ABB RAPID module: Module1.mod

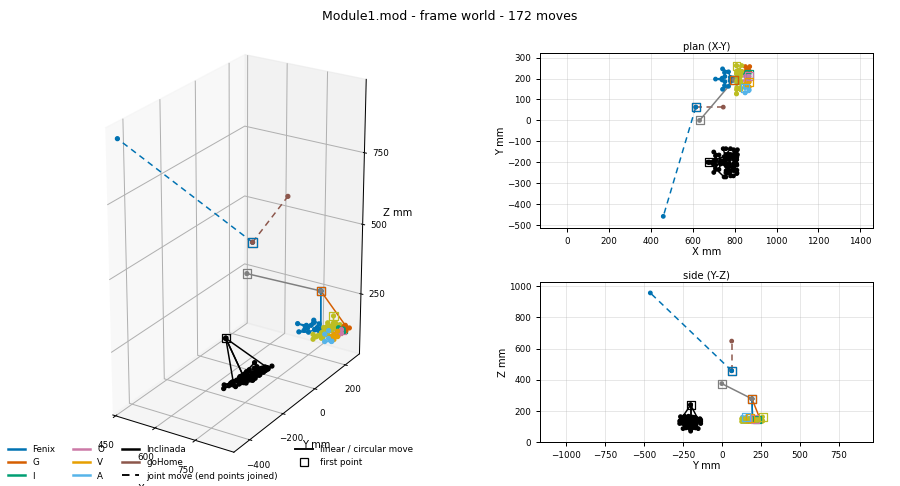
[picture p0: tool path of Module1.mod in frame world, 172 of 172 moves have a stored position in this frame; points joined in program order, loops and branches not executed]
MODULE Module1
    CONST robtarget Target_30:=[[-3.345189343,200,0],[0,0,1,0],[0,0,-1,1],[9E+09,9E+09,9E+09,9E+09,9E+09,9E+09]];
    CONST robtarget Target_20:=[[196.654810657,0,0],[0,0,1,0],[-1,-1,0,1],[9E+09,9E+09,9E+09,9E+09,9E+09,9E+09]];
    CONST robtarget Target_10:=[[811.652044776,0,588.439776326],[0.199367935,0,0.979924705,0],[0,0,0,0],[9E+09,9E+09,9E+09,9E+09,9E+09,9E+09]];
    CONST robtarget Target_40:=[[196.654810657,200,0],[0,0,1,0],[0,0,-1,1],[9E+09,9E+09,9E+09,9E+09,9E+09,9E+09]];
    CONST robtarget Target_50:=[[-3.345189343,0,0],[0,0,1,0],[-1,-1,0,1],[9E+09,9E+09,9E+09,9E+09,9E+09,9E+09]];
    CONST robtarget Home:=[[99.759101071,96.787006521,143.600305669],[0.000000093,0.707106794,-0.707106768,0.00000008],[0,-1,-1,0],[9E+09,9E+09,9E+09,9E+09,9E+09,9E+09]];
    CONST robtarget Target_110:=[[99.759,96.787,0],[0,-0.707106781,0.707106781,0],[0,-1,-1,0],[9E+09,9E+09,9E+09,9E+09,9E+09,9E+09]];
    CONST robtarget Target_140:=[[104.929185141,91.208348507,-1],[0,-0.707106781,0.707106781,0],[0,-1,-1,0],[9E+09,9E+09,9E+09,9E+09,9E+09,9E+09]];
    CONST robtarget Target_150:=[[107.828310564,78.545833086,-1],[0,-0.707106781,0.707106781,0],[0,-1,-1,0],[9E+09,9E+09,9E+09,9E+09,9E+09,9E+09]];
    CONST robtarget Target_160:=[[107.828310564,78.545833086,0],[0,-0.707106781,0.707106781,0],[0,-1,-1,0],[9E+09,9E+09,9E+09,9E+09,9E+09,9E+09]];
    CONST robtarget Target_170:=[[134.404345915,70.350066147,0],[0,-0.707106781,0.707106781,0],[0,-1,-1,0],[9E+09,9E+09,9E+09,9E+09,9E+09,9E+09]];
    CONST robtarget Target_180:=[[148.580115129,41.813525252,0],[0,-0.707106781,0.707106781,0],[0,-1,-1,0],[9E+09,9E+09,9E+09,9E+09,9E+09,9E+09]];
    CONST robtarget Target_190:=[[130.91133859,51.285461834,0],[0,-0.707106781,0.707106781,0],[0,-1,-1,0],[9E+09,9E+09,9E+09,9E+09,9E+09,9E+09]];
    CONST robtarget Target_200:=[[111.937087331,53.067189269,0],[0,-0.707106781,0.707106781,0],[0,-1,-1,0],[9E+09,9E+09,9E+09,9E+09,9E+09,9E+09]];
    CONST robtarget Target_210:=[[103.845690477,39.688183175,0],[0,-0.707106781,0.707106781,0],[0,-1,0,0],[9E+09,9E+09,9E+09,9E+09,9E+09,9E+09]];
    CONST robtarget Target_220:=[[99.759,8.211459743,0],[0,-0.707106781,0.707106781,0],[0,-1,0,0],[9E+09,9E+09,9E+09,9E+09,9E+09,9E+09]];
    CONST robtarget Target_230:=[[95.672309523,39.688183175,0],[0,-0.707106781,0.707106781,0],[0,-1,0,0],[9E+09,9E+09,9E+09,9E+09,9E+09,9E+09]];
    CONST robtarget Target_240:=[[87.580912669,53.067189269,0],[0,-0.707106781,0.707106781,0],[0,-1,0,0],[9E+09,9E+09,9E+09,9E+09,9E+09,9E+09]];
    CONST robtarget Target_250:=[[68.60666141,51.285461834,0],[0,-0.707106781,0.707106781,0],[0,-1,0,0],[9E+09,9E+09,9E+09,9E+09,9E+09,9E+09]];
    CONST robtarget Target_260:=[[50.937884871,41.813525252,0],[0,-0.707106781,0.707106781,0],[0,-1,0,0],[9E+09,9E+09,9E+09,9E+09,9E+09,9E+09]];
    CONST robtarget Target_270:=[[65.113654085,70.350066147,0],[0,-0.707106781,0.707106781,0],[0,-1,0,0],[9E+09,9E+09,9E+09,9E+09,9E+09,9E+09]];
    CONST robtarget Target_280:=[[91.689689436,78.545833086,0],[0,-0.707106781,0.707106781,0],[0,-1,-1,0],[9E+09,9E+09,9E+09,9E+09,9E+09,9E+09]];
    CONST robtarget Target_290:=[[94.588814859,91.208348507,0],[0,-0.707106781,0.707106781,0],[0,-1,-1,0],[9E+09,9E+09,9E+09,9E+09,9E+09,9E+09]];
    CONST robtarget Target_300:=[[99.759,96.787186115,0],[0,-0.707106781,0.707106781,0],[0,-1,-1,0],[9E+09,9E+09,9E+09,9E+09,9E+09,9E+09]];
    CONST robtarget Target_310:=[[51.434050484,162.594498178,0],[0,-0.707106781,0.707106781,0],[0,-1,-1,0],[9E+09,9E+09,9E+09,9E+09,9E+09,9E+09]];
    CONST robtarget Target_320:=[[64.567186307,162.594498178,0],[0,-0.707106781,0.707106781,0],[0,-1,-1,0],[9E+09,9E+09,9E+09,9E+09,9E+09,9E+09]];
    CONST robtarget Target_330:=[[63.433064042,150.856332741,0],[0,-0.707106781,0.707106781,0],[0,-1,-1,0],[9E+09,9E+09,9E+09,9E+09,9E+09,9E+09]];
    CONST robtarget Target_340:=[[40.013439281,150.867673964,0],[0,-0.707106781,0.707106781,0],[0,-1,-1,0],[9E+09,9E+09,9E+09,9E+09,9E+09,9E+09]];
    CONST robtarget Target_350:=[[40.013439281,171.554064067,0],[0,-0.707106781,0.707106781,0],[0,-1,-1,0],[9E+09,9E+09,9E+09,9E+09,9E+09,9E+09]];
    CONST robtarget Target_360:=[[63.410381597,171.588087735,0],[0,-0.707106781,0.707106781,0],[0,-1,-1,0],[9E+09,9E+09,9E+09,9E+09,9E+09,9E+09]];
    CONST robtarget Target_370:=[[64.567186307,167.539271251,0],[0,-0.707106781,0.707106781,0],[0,-1,-1,0],[9E+09,9E+09,9E+09,9E+09,9E+09,9E+09]];
    CONST robtarget Target_380:=[[67.932991772,167.539512506,10.290593582],[0.000000041,-0.707106747,0.707106815,0.000000103],[0,-1,-1,0],[9E+09,9E+09,9E+09,9E+09,9E+09,9E+09]];
    CONST robtarget Target_390:=[[73.897948354,167.539514704,10.290568716],[0.000000024,0.70710679,-0.707106772,-0.000000187],[0,-1,-1,0],[9E+09,9E+09,9E+09,9E+09,9E+09,9E+09]];
    CONST robtarget Target_410:=[[73.912353766,168.537298844,0],[0,-0.707106781,0.707106781,0],[0,-1,-1,0],[9E+09,9E+09,9E+09,9E+09,9E+09,9E+09]];
    CONST robtarget Target_400:=[[73.912353766,149.710869254,0],[0,-0.707106781,0.707106781,0],[0,-1,-1,0],[9E+09,9E+09,9E+09,9E+09,9E+09,9E+09]];
    CONST robtarget Target_420:=[[73.912362356,149.710913626,10.190706901],[0.000000042,0.707106789,-0.707106773,-0.000000141],[0,-1,-1,0],[9E+09,9E+09,9E+09,9E+09,9E+09,9E+09]];
    CONST robtarget Target_480:=[[86.637199295,167.641310207,13.160930267],[0.000000042,0.707106788,-0.707106775,-0.000000007],[0,-1,-1,0],[9E+09,9E+09,9E+09,9E+09,9E+09,9E+09]];
    CONST robtarget Target_470:=[[86.637205573,167.641342255,0],[0,-0.707106781,0.707106781,0],[0,-1,-1,0],[9E+09,9E+09,9E+09,9E+09,9E+09,9E+09]];
    CONST robtarget Target_440:=[[107.59578502,167.641342255,0],[0,-0.707106781,0.707106781,0],[0,-1,-1,0],[9E+09,9E+09,9E+09,9E+09,9E+09,9E+09]];
    CONST robtarget Target_450:=[[107.607126243,150.652190733,0],[0,-0.707106781,0.707106781,0],[0,-1,-1,0],[9E+09,9E+09,9E+09,9E+09,9E+09,9E+09]];
    CONST robtarget Target_460:=[[86.614523128,150.640849511,0],[0,-0.707106781,0.707106781,0],[0,-1,-1,0],[9E+09,9E+09,9E+09,9E+09,9E+09,9E+09]];
    CONST robtarget Target_530:=[[113.447892452,168.582709847,19.902538584],[0.000000053,0.707106797,-0.707106766,-0.000000049],[0,-1,-1,0],[9E+09,9E+09,9E+09,9E+09,9E+09,9E+09]];
    CONST robtarget Target_490:=[[113.447855905,168.582663735,0],[0,-0.707106781,0.707106781,0],[0,-1,-1,0],[9E+09,9E+09,9E+09,9E+09,9E+09,9E+09]];
    CONST robtarget Target_500:=[[124.335429644,149.710869254,0],[0,-0.707106781,0.707106781,0],[0,-1,-1,0],[9E+09,9E+09,9E+09,9E+09,9E+09,9E+09]];
    CONST robtarget Target_520:=[[127.035,149.711,0],[0,-0.707106781,0.707106781,0],[0,-1,-1,0],[9E+09,9E+09,9E+09,9E+09,9E+09,9E+09]];
    CONST robtarget Target_510:=[[137.377835685,168.582663735,0],[0,-0.707106781,0.707106781,0],[0,-1,-1,0],[9E+09,9E+09,9E+09,9E+09,9E+09,9E+09]];
    CONST robtarget Target_540:=[[137.377791379,168.582717891,19.385142962],[0.000000048,0.707106782,-0.70710678,-0.00000004],[0,-1,-1,0],[9E+09,9E+09,9E+09,9E+09,9E+09,9E+09]];
    CONST robtarget Target_590:=[[139.645827027,149.710937127,28.980061356],[-0.000000039,0.707106799,-0.707106764,-0.00000025],[0,-1,-1,0],[9E+09,9E+09,9E+09,9E+09,9E+09,9E+09]];
    CONST robtarget Target_550:=[[139.646080214,149.710869254,0],[0,-0.707106781,0.707106781,0],[0,-1,-1,0],[9E+09,9E+09,9E+09,9E+09,9E+09,9E+09]];
    CONST robtarget Target_560:=[[150.556336398,168.582663735,0],[0,-0.707106781,0.707106781,0],[0,-1,-1,0],[9E+09,9E+09,9E+09,9E+09,9E+09,9E+09]];
    CONST robtarget Target_570:=[[153.822608519,168.582663735,0],[0,-0.707106781,0.707106781,0],[0,-1,-1,0],[9E+09,9E+09,9E+09,9E+09,9E+09,9E+09]];
    CONST robtarget Target_580:=[[165.005054047,149.710869254,0],[0,-0.707106781,0.707106781,0],[0,-1,-1,0],[9E+09,9E+09,9E+09,9E+09,9E+09,9E+09]];
    CONST robtarget Target_600:=[[165.005120388,149.710943698,27.340042804],[0.000000095,0.707106812,-0.707106751,0.000000059],[0,-1,-1,0],[9E+09,9E+09,9E+09,9E+09,9E+09,9E+09]];
    CONST robtarget Home_3:=[[99.759101071,96.787006521,143.600305669],[0.000000093,0.707106794,-0.707106768,0.00000008],[1,1,0,7],[9E+09,9E+09,9E+09,9E+09,9E+09,9E+09]];
    CONST robtarget Target_110_3:=[[99.759,96.787,0],[0,-0.707106781,0.707106781,0],[1,1,-1,7],[9E+09,9E+09,9E+09,9E+09,9E+09,9E+09]];
    CONST robtarget Target_140_3:=[[104.929185141,91.208348507,-1],[0,-0.707106781,0.707106781,0],[1,1,-1,7],[9E+09,9E+09,9E+09,9E+09,9E+09,9E+09]];
    CONST robtarget Target_150_3:=[[107.828310564,78.545833086,-1],[0,-0.707106781,0.707106781,0],[1,1,-1,7],[9E+09,9E+09,9E+09,9E+09,9E+09,9E+09]];
    CONST robtarget Target_160_3:=[[107.828310564,78.545833086,0],[0,-0.707106781,0.707106781,0],[1,1,-1,7],[9E+09,9E+09,9E+09,9E+09,9E+09,9E+09]];
    CONST robtarget Target_170_3:=[[134.404345915,70.350066147,0],[0,-0.707106781,0.707106781,0],[1,1,-1,7],[9E+09,9E+09,9E+09,9E+09,9E+09,9E+09]];
    CONST robtarget Target_180_3:=[[148.580115129,41.813525252,0],[0,-0.707106781,0.707106781,0],[1,1,-1,7],[9E+09,9E+09,9E+09,9E+09,9E+09,9E+09]];
    CONST robtarget Target_190_3:=[[130.91133859,51.285461834,0],[0,-0.707106781,0.707106781,0],[1,1,-1,7],[9E+09,9E+09,9E+09,9E+09,9E+09,9E+09]];
    CONST robtarget Target_200_3:=[[111.937087331,53.067189269,0],[0,-0.707106781,0.707106781,0],[1,1,-1,7],[9E+09,9E+09,9E+09,9E+09,9E+09,9E+09]];
    CONST robtarget Target_210_3:=[[103.845690477,39.688183175,0],[0,-0.707106781,0.707106781,0],[1,1,-1,7],[9E+09,9E+09,9E+09,9E+09,9E+09,9E+09]];
    CONST robtarget Target_220_3:=[[99.759,8.211459743,0],[0,-0.707106781,0.707106781,0],[0,0,-1,7],[9E+09,9E+09,9E+09,9E+09,9E+09,9E+09]];
    CONST robtarget Target_230_3:=[[95.672309523,39.688183175,0],[0,-0.707106781,0.707106781,0],[1,1,-1,7],[9E+09,9E+09,9E+09,9E+09,9E+09,9E+09]];
    CONST robtarget Target_240_3:=[[87.580912669,53.067189269,0],[0,-0.707106781,0.707106781,0],[1,1,-1,7],[9E+09,9E+09,9E+09,9E+09,9E+09,9E+09]];
    CONST robtarget Target_250_3:=[[68.60666141,51.285461834,0],[0,-0.707106781,0.707106781,0],[1,1,-1,7],[9E+09,9E+09,9E+09,9E+09,9E+09,9E+09]];
    CONST robtarget Target_260_3:=[[50.937884871,41.813525252,0],[0,-0.707106781,0.707106781,0],[1,1,-1,7],[9E+09,9E+09,9E+09,9E+09,9E+09,9E+09]];
    CONST robtarget Target_270_3:=[[65.113654085,70.350066147,0],[0,-0.707106781,0.707106781,0],[1,1,-1,7],[9E+09,9E+09,9E+09,9E+09,9E+09,9E+09]];
    CONST robtarget Target_280_3:=[[91.689689436,78.545833086,0],[0,-0.707106781,0.707106781,0],[1,1,-1,7],[9E+09,9E+09,9E+09,9E+09,9E+09,9E+09]];
    CONST robtarget Target_290_3:=[[94.588814859,91.208348507,0],[0,-0.707106781,0.707106781,0],[1,1,-1,7],[9E+09,9E+09,9E+09,9E+09,9E+09,9E+09]];
    CONST robtarget Target_300_3:=[[99.759,96.787186115,0],[0,-0.707106781,0.707106781,0],[1,1,-1,7],[9E+09,9E+09,9E+09,9E+09,9E+09,9E+09]];
    CONST robtarget Target_310_3:=[[51.434050484,162.594498178,0],[0,-0.707106781,0.707106781,0],[1,1,-1,7],[9E+09,9E+09,9E+09,9E+09,9E+09,9E+09]];
    CONST robtarget Target_320_3:=[[64.567186307,162.594498178,0],[0,-0.707106781,0.707106781,0],[1,1,-1,7],[9E+09,9E+09,9E+09,9E+09,9E+09,9E+09]];
    CONST robtarget Target_330_3:=[[63.433064042,150.856332741,0],[0,-0.707106781,0.707106781,0],[1,1,-1,7],[9E+09,9E+09,9E+09,9E+09,9E+09,9E+09]];
    CONST robtarget Target_340_3:=[[40.013439281,150.867673964,0],[0,-0.707106781,0.707106781,0],[1,1,-1,7],[9E+09,9E+09,9E+09,9E+09,9E+09,9E+09]];
    CONST robtarget Target_350_3:=[[40.013439281,171.554064067,0],[0,-0.707106781,0.707106781,0],[1,1,-1,7],[9E+09,9E+09,9E+09,9E+09,9E+09,9E+09]];
    CONST robtarget Target_360_3:=[[63.410381597,171.588087735,0],[0,-0.707106781,0.707106781,0],[1,1,-1,7],[9E+09,9E+09,9E+09,9E+09,9E+09,9E+09]];
    CONST robtarget Target_370_3:=[[64.567186307,167.539271251,0],[0,-0.707106781,0.707106781,0],[1,1,-1,7],[9E+09,9E+09,9E+09,9E+09,9E+09,9E+09]];
    CONST robtarget Target_380_3:=[[67.932991772,167.539512506,10.290593582],[0.000000041,-0.707106747,0.707106815,0.000000103],[1,1,-1,7],[9E+09,9E+09,9E+09,9E+09,9E+09,9E+09]];
    CONST robtarget Target_390_3:=[[73.897948354,167.539514704,10.290568716],[0.000000024,0.70710679,-0.707106772,-0.000000187],[1,1,-1,7],[9E+09,9E+09,9E+09,9E+09,9E+09,9E+09]];
    CONST robtarget Target_410_3:=[[73.912353766,168.537298844,0],[0,-0.707106781,0.707106781,0],[1,1,-1,7],[9E+09,9E+09,9E+09,9E+09,9E+09,9E+09]];
    CONST robtarget Target_400_3:=[[73.912353766,149.710869254,0],[0,-0.707106781,0.707106781,0],[1,1,-1,7],[9E+09,9E+09,9E+09,9E+09,9E+09,9E+09]];
    CONST robtarget Target_420_3:=[[73.912362356,149.710913626,10.190706901],[0.000000042,0.707106789,-0.707106773,-0.000000141],[1,1,-1,7],[9E+09,9E+09,9E+09,9E+09,9E+09,9E+09]];
    CONST robtarget Target_480_3:=[[86.637199295,167.641310207,13.160930267],[0.000000042,0.707106788,-0.707106775,-0.000000007],[1,1,-1,7],[9E+09,9E+09,9E+09,9E+09,9E+09,9E+09]];
    CONST robtarget Target_470_3:=[[86.637205573,167.641342255,0],[0,-0.707106781,0.707106781,0],[1,1,-1,7],[9E+09,9E+09,9E+09,9E+09,9E+09,9E+09]];
    CONST robtarget Target_440_3:=[[107.59578502,167.641342255,0],[0,-0.707106781,0.707106781,0],[1,1,0,7],[9E+09,9E+09,9E+09,9E+09,9E+09,9E+09]];
    CONST robtarget Target_450_3:=[[107.607126243,150.652190733,0],[0,-0.707106781,0.707106781,0],[1,1,-1,7],[9E+09,9E+09,9E+09,9E+09,9E+09,9E+09]];
    CONST robtarget Target_460_3:=[[86.614523128,150.640849511,0],[0,-0.707106781,0.707106781,0],[1,1,-1,7],[9E+09,9E+09,9E+09,9E+09,9E+09,9E+09]];
    CONST robtarget Target_530_3:=[[113.447892452,168.582709847,19.902538584],[0.000000053,0.707106797,-0.707106766,-0.000000049],[1,1,0,7],[9E+09,9E+09,9E+09,9E+09,9E+09,9E+09]];
    CONST robtarget Target_490_3:=[[113.447855905,168.582663735,0],[0,-0.707106781,0.707106781,0],[1,1,0,7],[9E+09,9E+09,9E+09,9E+09,9E+09,9E+09]];
    CONST robtarget Target_500_3:=[[124.335429644,149.710869254,0],[0,-0.707106781,0.707106781,0],[1,1,0,7],[9E+09,9E+09,9E+09,9E+09,9E+09,9E+09]];
    CONST robtarget Target_520_3:=[[127.035,149.711,0],[0,-0.707106781,0.707106781,0],[1,1,0,7],[9E+09,9E+09,9E+09,9E+09,9E+09,9E+09]];
    CONST robtarget Target_510_3:=[[137.377835685,168.582663735,0],[0,-0.707106781,0.707106781,0],[1,1,0,7],[9E+09,9E+09,9E+09,9E+09,9E+09,9E+09]];
    CONST robtarget Target_540_3:=[[137.377791379,168.582717891,19.385142962],[0.000000048,0.707106782,-0.70710678,-0.00000004],[1,1,0,7],[9E+09,9E+09,9E+09,9E+09,9E+09,9E+09]];
    CONST robtarget Target_590_3:=[[139.645827027,149.710937127,28.980061356],[-0.000000039,0.707106799,-0.707106764,-0.00000025],[1,1,0,7],[9E+09,9E+09,9E+09,9E+09,9E+09,9E+09]];
    CONST robtarget Target_550_3:=[[139.646080214,149.710869254,0],[0,-0.707106781,0.707106781,0],[1,1,0,7],[9E+09,9E+09,9E+09,9E+09,9E+09,9E+09]];
    CONST robtarget Target_560_3:=[[150.556336398,168.582663735,0],[0,-0.707106781,0.707106781,0],[1,1,0,7],[9E+09,9E+09,9E+09,9E+09,9E+09,9E+09]];
    CONST robtarget Target_570_3:=[[153.822608519,168.582663735,0],[0,-0.707106781,0.707106781,0],[1,1,0,7],[9E+09,9E+09,9E+09,9E+09,9E+09,9E+09]];
    CONST robtarget Target_580_3:=[[165.005054047,149.710869254,0],[0,-0.707106781,0.707106781,0],[1,1,0,7],[9E+09,9E+09,9E+09,9E+09,9E+09,9E+09]];
    CONST robtarget Target_600_3:=[[165.005120388,149.710943698,27.340042804],[0.000000095,0.707106812,-0.707106751,0.000000059],[1,1,0,7],[9E+09,9E+09,9E+09,9E+09,9E+09,9E+09]];
    CONST robtarget Target_650:=[[631.875981178,0,375.874287303],[0.171236408,0,-0.985229969,0],[0,0,0,0],[9E+09,9E+09,9E+09,9E+09,9E+09,9E+09]];
    CONST robtarget Target_660:=[[35.046842978,108.443166881,26.254106583],[0,-0.707106781,0.707106781,0],[0,-1,-1,0],[9E+09,9E+09,9E+09,9E+09,9E+09,9E+09]];
    CONST robtarget Target_720:=[[35.047,108.443,0],[0,-0.707106781,0.707106781,0],[0,-1,-1,0],[9E+09,9E+09,9E+09,9E+09,9E+09,9E+09]];
    CONST robtarget Target_670:=[[35.046842978,133.443166881,0],[0,-0.707106781,0.707106781,0],[0,-1,-1,0],[9E+09,9E+09,9E+09,9E+09,9E+09,9E+09]];
    CONST robtarget Target_680:=[[56.373272958,116.727190549,0],[0,-0.707106781,0.707106781,0],[0,-1,-1,0],[9E+09,9E+09,9E+09,9E+09,9E+09,9E+09]];
    CONST robtarget Target_700:=[[62.660255206,108.443166881,0],[0,-0.707106781,0.707106781,0],[0,-1,-1,0],[9E+09,9E+09,9E+09,9E+09,9E+09,9E+09]];
    CONST robtarget Target_690:=[[62.660255206,133.443166881,0],[0,-0.707106781,0.707106781,0],[0,-1,-1,0],[9E+09,9E+09,9E+09,9E+09,9E+09,9E+09]];
    CONST robtarget Target_710:=[[62.660295778,133.257702122,17.408483113],[0.000000021,-0.707106766,0.707106797,0.000000049],[0,-1,-1,0],[9E+09,9E+09,9E+09,9E+09,9E+09,9E+09]];
    CONST robtarget Target_750:=[[73.779599663,128.906804208,17.663729092],[0.000000032,-0.70710677,0.707106793,0.000000042],[0,-1,-1,0],[9E+09,9E+09,9E+09,9E+09,9E+09,9E+09]];
    CONST robtarget Target_740:=[[73.779584595,128.906677729,0],[0,-0.707106781,0.707106781,0],[0,-1,-1,0],[9E+09,9E+09,9E+09,9E+09,9E+09,9E+09]];
    CONST robtarget Target_730:=[[73.779584595,108.443166881,0],[0,-0.707106781,0.707106781,0],[0,-1,-1,0],[9E+09,9E+09,9E+09,9E+09,9E+09,9E+09]];
    CONST robtarget Target_760:=[[73.779598222,108.443224437,17.731547844],[0.000000044,0.707106796,-0.707106766,-0.000000021],[0,-1,-1,0],[9E+09,9E+09,9E+09,9E+09,9E+09,9E+09]];
    CONST robtarget Target_830:=[[108.64148442,113.300223581,16.844032683],[0.000000008,0.707106783,-0.707106779,-0.000000028],[0,-1,-1,0],[9E+09,9E+09,9E+09,9E+09,9E+09,9E+09]];
    CONST robtarget Target_770:=[[108.641517534,113.300168853,0],[0,-0.707106781,0.707106781,0],[0,-1,-1,0],[9E+09,9E+09,9E+09,9E+09,9E+09,9E+09]];
    CONST robtarget Target_780:=[[107.593687159,109.466342423,0],[0,-0.707106781,0.707106781,0],[0,-1,-1,0],[9E+09,9E+09,9E+09,9E+09,9E+09,9E+09]];
    CONST robtarget Target_790:=[[87.573963293,109.429360175,0],[0,-0.707106781,0.707106781,0],[0,-1,-1,0],[9E+09,9E+09,9E+09,9E+09,9E+09,9E+09]];
    CONST robtarget Target_800:=[[87.586290709,127.945139267,0],[0,-0.707106781,0.707106781,0],[0,-1,-1,0],[9E+09,9E+09,9E+09,9E+09,9E+09,9E+09]];
    CONST robtarget Target_810:=[[107.593687159,127.932811851,0],[0,-0.707106781,0.707106781,0],[0,-1,-1,0],[9E+09,9E+09,9E+09,9E+09,9E+09,9E+09]];
    CONST robtarget Target_820:=[[108.641517534,124.074330589,0],[0,-0.707106781,0.707106781,0],[0,-1,-1,0],[9E+09,9E+09,9E+09,9E+09,9E+09,9E+09]];
    CONST robtarget Target_840:=[[108.641489854,124.074419597,17.530850048],[0.000000038,0.707106785,-0.707106778,-0.000000018],[0,-1,-1,0],[9E+09,9E+09,9E+09,9E+09,9E+09,9E+09]];
    CONST robtarget Target_900:=[[117.443278694,127.932797325,17.936531586],[-0.000000069,-0.707106731,0.707106831,0.000000105],[0,-1,-1,0],[9E+09,9E+09,9E+09,9E+09,9E+09,9E+09]];
    CONST robtarget Target_860:=[[117.443292682,127.932811851,0],[0,-0.707106781,0.707106781,0],[0,-1,-1,0],[9E+09,9E+09,9E+09,9E+09,9E+09,9E+09]];
    CONST robtarget Target_870:=[[140.224357771,127.932811851,0],[0,-0.707106781,0.707106781,0],[0,-1,-1,0],[9E+09,9E+09,9E+09,9E+09,9E+09,9E+09]];
    CONST robtarget Target_880:=[[140.236685187,109.466342423,0],[0,-0.707106781,0.707106781,0],[0,-1,-1,0],[9E+09,9E+09,9E+09,9E+09,9E+09,9E+09]];
    CONST robtarget Target_890:=[[117.418637849,109.454015007,0],[0,-0.707106781,0.707106781,0],[0,-1,-1,0],[9E+09,9E+09,9E+09,9E+09,9E+09,9E+09]];
    CONST robtarget Target_940:=[[150.283504114,128.956035202,17.783725507],[0,-0.707106781,0.707106781,0],[0,-1,-1,0],[9E+09,9E+09,9E+09,9E+09,9E+09,9E+09]];
    CONST robtarget Target_910:=[[150.283529368,128.955987394,0],[0,-0.707106781,0.707106781,0],[0,-1,-1,0],[9E+09,9E+09,9E+09,9E+09,9E+09,9E+09]];
    CONST robtarget Target_920:=[[150.283529368,108.443166881,0],[0,-0.707106781,0.707106781,0],[0,-1,-1,0],[9E+09,9E+09,9E+09,9E+09,9E+09,9E+09]];
    CONST robtarget Target_930:=[[170.106014575,108.443166881,0],[0,-0.707106781,0.707106781,0],[0,-1,-1,0],[9E+09,9E+09,9E+09,9E+09,9E+09,9E+09]];
    CONST robtarget Target_950:=[[170.105997965,108.443230949,17.745858799],[0.000000043,-0.707106776,0.707106786,0.000000052],[0,-1,-1,0],[9E+09,9E+09,9E+09,9E+09,9E+09,9E+09]];
    CONST robtarget Target_960:=[[51.434000123,162.594505433,12.553324918],[0.000000004,-0.707106757,0.707106805,0.000000033],[0,-1,-1,0],[9E+09,9E+09,9E+09,9E+09,9E+09,9E+09]];
    CONST robtarget Home_2:=[[99.759101071,96.787006521,143.600305669],[0.000000093,0.707106794,-0.707106768,0.00000008],[-1,-1,0,1],[9E+09,9E+09,9E+09,9E+09,9E+09,9E+09]];
    CONST robtarget Target_110_2:=[[99.759,96.787,0],[0,-0.707106781,0.707106781,0],[-1,-1,0,1],[9E+09,9E+09,9E+09,9E+09,9E+09,9E+09]];
    CONST robtarget Target_140_2:=[[104.929185141,91.208348507,-1],[0,-0.707106781,0.707106781,0],[-1,-1,0,1],[9E+09,9E+09,9E+09,9E+09,9E+09,9E+09]];
    CONST robtarget Target_150_2:=[[107.828310564,78.545833086,-1],[0,-0.707106781,0.707106781,0],[-1,-1,0,1],[9E+09,9E+09,9E+09,9E+09,9E+09,9E+09]];
    CONST robtarget Target_160_2:=[[107.828310564,78.545833086,0],[0,-0.707106781,0.707106781,0],[-1,-1,0,1],[9E+09,9E+09,9E+09,9E+09,9E+09,9E+09]];
    CONST robtarget Target_170_2:=[[134.404345915,70.350066147,0],[0,-0.707106781,0.707106781,0],[-1,-1,0,1],[9E+09,9E+09,9E+09,9E+09,9E+09,9E+09]];
    CONST robtarget Target_180_2:=[[148.580115129,41.813525252,0],[0,-0.707106781,0.707106781,0],[-1,-1,0,1],[9E+09,9E+09,9E+09,9E+09,9E+09,9E+09]];
    CONST robtarget Target_190_2:=[[130.91133859,51.285461834,0],[0,-0.707106781,0.707106781,0],[-1,-1,0,1],[9E+09,9E+09,9E+09,9E+09,9E+09,9E+09]];
    CONST robtarget Target_200_2:=[[111.937087331,53.067189269,0],[0,-0.707106781,0.707106781,0],[-1,-1,-1,1],[9E+09,9E+09,9E+09,9E+09,9E+09,9E+09]];
    CONST robtarget Target_210_2:=[[103.845690477,39.688183175,0],[0,-0.707106781,0.707106781,0],[-1,-1,-1,1],[9E+09,9E+09,9E+09,9E+09,9E+09,9E+09]];
    CONST robtarget Target_220_2:=[[99.759,8.211459743,0],[0,-0.707106781,0.707106781,0],[-1,-1,-1,1],[9E+09,9E+09,9E+09,9E+09,9E+09,9E+09]];
    CONST robtarget Target_230_2:=[[95.672309523,39.688183175,0],[0,-0.707106781,0.707106781,0],[-1,-1,-1,1],[9E+09,9E+09,9E+09,9E+09,9E+09,9E+09]];
    CONST robtarget Target_240_2:=[[87.580912669,53.067189269,0],[0,-0.707106781,0.707106781,0],[-1,-1,-1,1],[9E+09,9E+09,9E+09,9E+09,9E+09,9E+09]];
    CONST robtarget Target_250_2:=[[68.60666141,51.285461834,0],[0,-0.707106781,0.707106781,0],[-1,-1,-1,1],[9E+09,9E+09,9E+09,9E+09,9E+09,9E+09]];
    CONST robtarget Target_260_2:=[[50.937884871,41.813525252,0],[0,-0.707106781,0.707106781,0],[-1,-1,-1,1],[9E+09,9E+09,9E+09,9E+09,9E+09,9E+09]];
    CONST robtarget Target_270_2:=[[65.113654085,70.350066147,0],[0,-0.707106781,0.707106781,0],[-1,-1,-1,1],[9E+09,9E+09,9E+09,9E+09,9E+09,9E+09]];
    CONST robtarget Target_280_2:=[[91.689689436,78.545833086,0],[0,-0.707106781,0.707106781,0],[-1,-1,0,1],[9E+09,9E+09,9E+09,9E+09,9E+09,9E+09]];
    CONST robtarget Target_290_2:=[[94.588814859,91.208348507,0],[0,-0.707106781,0.707106781,0],[-1,-1,0,1],[9E+09,9E+09,9E+09,9E+09,9E+09,9E+09]];
    CONST robtarget Target_300_2:=[[99.759,96.787186115,0],[0,-0.707106781,0.707106781,0],[-1,-1,0,1],[9E+09,9E+09,9E+09,9E+09,9E+09,9E+09]];
    CONST robtarget Target_310_2:=[[51.434050484,162.594498178,0],[0,-0.707106781,0.707106781,0],[-1,-1,0,1],[9E+09,9E+09,9E+09,9E+09,9E+09,9E+09]];
    CONST robtarget Target_320_2:=[[64.567186307,162.594498178,0],[0,-0.707106781,0.707106781,0],[-1,-1,0,1],[9E+09,9E+09,9E+09,9E+09,9E+09,9E+09]];
    CONST robtarget Target_330_2:=[[63.433064042,150.856332741,0],[0,-0.707106781,0.707106781,0],[-1,-1,0,1],[9E+09,9E+09,9E+09,9E+09,9E+09,9E+09]];
    CONST robtarget Target_340_2:=[[40.013439281,150.867673964,0],[0,-0.707106781,0.707106781,0],[-1,-1,0,1],[9E+09,9E+09,9E+09,9E+09,9E+09,9E+09]];
    CONST robtarget Target_350_2:=[[40.013439281,171.554064067,0],[0,-0.707106781,0.707106781,0],[-1,-1,0,1],[9E+09,9E+09,9E+09,9E+09,9E+09,9E+09]];
    CONST robtarget Target_360_2:=[[63.410381597,171.588087735,0],[0,-0.707106781,0.707106781,0],[-1,-1,0,1],[9E+09,9E+09,9E+09,9E+09,9E+09,9E+09]];
    CONST robtarget Target_370_2:=[[64.567186307,167.539271251,0],[0,-0.707106781,0.707106781,0],[-1,-1,0,1],[9E+09,9E+09,9E+09,9E+09,9E+09,9E+09]];
    CONST robtarget Target_380_2:=[[67.932991772,167.539512506,10.290593582],[0.000000041,-0.707106747,0.707106815,0.000000103],[-1,-1,0,1],[9E+09,9E+09,9E+09,9E+09,9E+09,9E+09]];
    CONST robtarget Target_390_2:=[[73.897948354,167.539514704,10.290568716],[0.000000024,0.70710679,-0.707106772,-0.000000187],[-1,-1,0,1],[9E+09,9E+09,9E+09,9E+09,9E+09,9E+09]];
    CONST robtarget Target_410_2:=[[73.912353766,168.537298844,0],[0,-0.707106781,0.707106781,0],[-1,-1,0,1],[9E+09,9E+09,9E+09,9E+09,9E+09,9E+09]];
    CONST robtarget Target_400_2:=[[73.912353766,149.710869254,0],[0,-0.707106781,0.707106781,0],[-1,-1,0,1],[9E+09,9E+09,9E+09,9E+09,9E+09,9E+09]];
    CONST robtarget Target_420_2:=[[73.912362356,149.710913626,10.190706901],[0.000000042,0.707106789,-0.707106773,-0.000000141],[-1,-1,0,1],[9E+09,9E+09,9E+09,9E+09,9E+09,9E+09]];
    CONST robtarget Target_480_2:=[[86.637199295,167.641310207,13.160930267],[0.000000042,0.707106788,-0.707106775,-0.000000007],[-1,-1,0,1],[9E+09,9E+09,9E+09,9E+09,9E+09,9E+09]];
    CONST robtarget Target_470_2:=[[86.637205573,167.641342255,0],[0,-0.707106781,0.707106781,0],[-1,-1,0,1],[9E+09,9E+09,9E+09,9E+09,9E+09,9E+09]];
    CONST robtarget Target_440_2:=[[107.59578502,167.641342255,0],[0,-0.707106781,0.707106781,0],[-1,-1,0,1],[9E+09,9E+09,9E+09,9E+09,9E+09,9E+09]];
    CONST robtarget Target_450_2:=[[107.607126243,150.652190733,0],[0,-0.707106781,0.707106781,0],[-1,-1,0,1],[9E+09,9E+09,9E+09,9E+09,9E+09,9E+09]];
    CONST robtarget Target_460_2:=[[86.614523128,150.640849511,0],[0,-0.707106781,0.707106781,0],[-1,-1,0,1],[9E+09,9E+09,9E+09,9E+09,9E+09,9E+09]];
    CONST robtarget Target_530_2:=[[113.447892452,168.582709847,19.902538584],[0.000000053,0.707106797,-0.707106766,-0.000000049],[-1,-1,0,1],[9E+09,9E+09,9E+09,9E+09,9E+09,9E+09]];
    CONST robtarget Target_490_2:=[[113.447855905,168.582663735,0],[0,-0.707106781,0.707106781,0],[-1,-1,0,1],[9E+09,9E+09,9E+09,9E+09,9E+09,9E+09]];
    CONST robtarget Target_500_2:=[[124.335429644,149.710869254,0],[0,-0.707106781,0.707106781,0],[-1,-1,0,1],[9E+09,9E+09,9E+09,9E+09,9E+09,9E+09]];
    CONST robtarget Target_520_2:=[[127.035,149.711,0],[0,-0.707106781,0.707106781,0],[-1,-1,0,1],[9E+09,9E+09,9E+09,9E+09,9E+09,9E+09]];
    CONST robtarget Target_510_2:=[[137.377835685,168.582663735,0],[0,-0.707106781,0.707106781,0],[-1,-1,0,1],[9E+09,9E+09,9E+09,9E+09,9E+09,9E+09]];
    CONST robtarget Target_540_2:=[[137.377791379,168.582717891,19.385142962],[0.000000048,0.707106782,-0.70710678,-0.00000004],[-1,-1,0,1],[9E+09,9E+09,9E+09,9E+09,9E+09,9E+09]];
    CONST robtarget Target_590_2:=[[139.645827027,149.710937127,28.980061356],[-0.000000039,0.707106799,-0.707106764,-0.00000025],[-1,-1,0,1],[9E+09,9E+09,9E+09,9E+09,9E+09,9E+09]];
    CONST robtarget Target_550_2:=[[139.646080214,149.710869254,0],[0,-0.707106781,0.707106781,0],[-1,-1,0,1],[9E+09,9E+09,9E+09,9E+09,9E+09,9E+09]];
    CONST robtarget Target_560_2:=[[150.556336398,168.582663735,0],[0,-0.707106781,0.707106781,0],[-1,-1,0,1],[9E+09,9E+09,9E+09,9E+09,9E+09,9E+09]];
    CONST robtarget Target_570_2:=[[153.822608519,168.582663735,0],[0,-0.707106781,0.707106781,0],[-1,-1,0,1],[9E+09,9E+09,9E+09,9E+09,9E+09,9E+09]];
    CONST robtarget Target_580_2:=[[165.005054047,149.710869254,0],[0,-0.707106781,0.707106781,0],[-1,-1,0,1],[9E+09,9E+09,9E+09,9E+09,9E+09,9E+09]];
    CONST robtarget Target_600_2:=[[165.005120388,149.710943698,27.340042804],[0.000000095,0.707106812,-0.707106751,0.000000059],[-1,-1,0,1],[9E+09,9E+09,9E+09,9E+09,9E+09,9E+09]];
    CONST robtarget Target_660_2:=[[35.046842978,108.443166881,26.254106583],[0,-0.707106781,0.707106781,0],[-1,-1,0,1],[9E+09,9E+09,9E+09,9E+09,9E+09,9E+09]];
    CONST robtarget Target_720_2:=[[35.047,108.443,0],[0,-0.707106781,0.707106781,0],[-1,-1,0,1],[9E+09,9E+09,9E+09,9E+09,9E+09,9E+09]];
    CONST robtarget Target_670_2:=[[35.046842978,133.443166881,0],[0,-0.707106781,0.707106781,0],[-1,-1,0,1],[9E+09,9E+09,9E+09,9E+09,9E+09,9E+09]];
    CONST robtarget Target_700_2:=[[62.660255206,108.443166881,0],[0,-0.707106781,0.707106781,0],[-1,-1,0,1],[9E+09,9E+09,9E+09,9E+09,9E+09,9E+09]];
    CONST robtarget Target_690_2:=[[62.660255206,133.443166881,0],[0,-0.707106781,0.707106781,0],[-1,-1,0,1],[9E+09,9E+09,9E+09,9E+09,9E+09,9E+09]];
    CONST robtarget Target_710_2:=[[62.660295778,133.257702122,17.408483113],[0.000000021,-0.707106766,0.707106797,0.000000049],[-1,-1,0,1],[9E+09,9E+09,9E+09,9E+09,9E+09,9E+09]];
    CONST robtarget Target_750_2:=[[73.779599663,128.906804208,17.663729092],[0.000000032,-0.70710677,0.707106793,0.000000042],[-1,-1,0,1],[9E+09,9E+09,9E+09,9E+09,9E+09,9E+09]];
    CONST robtarget Target_740_2:=[[73.779584595,128.906677729,0],[0,-0.707106781,0.707106781,0],[-1,-1,0,1],[9E+09,9E+09,9E+09,9E+09,9E+09,9E+09]];
    CONST robtarget Target_730_2:=[[73.779584595,108.443166881,0],[0,-0.707106781,0.707106781,0],[-1,-1,0,1],[9E+09,9E+09,9E+09,9E+09,9E+09,9E+09]];
    CONST robtarget Target_760_2:=[[73.779598222,108.443224437,17.731547844],[0.000000044,0.707106796,-0.707106766,-0.000000021],[-1,-1,0,1],[9E+09,9E+09,9E+09,9E+09,9E+09,9E+09]];
    CONST robtarget Target_830_2:=[[108.64148442,113.300223581,16.844032683],[0.000000008,0.707106783,-0.707106779,-0.000000028],[-1,-1,0,1],[9E+09,9E+09,9E+09,9E+09,9E+09,9E+09]];
    CONST robtarget Target_770_2:=[[108.641517534,113.300168853,0],[0,-0.707106781,0.707106781,0],[-1,-1,0,1],[9E+09,9E+09,9E+09,9E+09,9E+09,9E+09]];
    CONST robtarget Target_780_2:=[[107.593687159,109.466342423,0],[0,-0.707106781,0.707106781,0],[-1,-1,0,1],[9E+09,9E+09,9E+09,9E+09,9E+09,9E+09]];
    CONST robtarget Target_790_2:=[[87.573963293,109.429360175,0],[0,-0.707106781,0.707106781,0],[-1,-1,0,1],[9E+09,9E+09,9E+09,9E+09,9E+09,9E+09]];
    CONST robtarget Target_800_2:=[[87.586290709,127.945139267,0],[0,-0.707106781,0.707106781,0],[-1,-1,0,1],[9E+09,9E+09,9E+09,9E+09,9E+09,9E+09]];
    CONST robtarget Target_810_2:=[[107.593687159,127.932811851,0],[0,-0.707106781,0.707106781,0],[-1,-1,0,1],[9E+09,9E+09,9E+09,9E+09,9E+09,9E+09]];
    CONST robtarget Target_820_2:=[[108.641517534,124.074330589,0],[0,-0.707106781,0.707106781,0],[-1,-1,0,1],[9E+09,9E+09,9E+09,9E+09,9E+09,9E+09]];
    CONST robtarget Target_840_2:=[[108.641489854,124.074419597,17.530850048],[0.000000038,0.707106785,-0.707106778,-0.000000018],[-1,-1,0,1],[9E+09,9E+09,9E+09,9E+09,9E+09,9E+09]];
    CONST robtarget Target_900_2:=[[117.443278694,127.932797325,17.936531586],[-0.000000069,-0.707106731,0.707106831,0.000000105],[-1,-1,0,1],[9E+09,9E+09,9E+09,9E+09,9E+09,9E+09]];
    CONST robtarget Target_860_3:=[[117.443292682,127.932811851,0],[0,-0.707106781,0.707106781,0],[-1,-1,0,1],[9E+09,9E+09,9E+09,9E+09,9E+09,9E+09]];
    CONST robtarget Target_870_2:=[[140.224357771,127.932811851,0],[0,-0.707106781,0.707106781,0],[-1,-1,0,1],[9E+09,9E+09,9E+09,9E+09,9E+09,9E+09]];
    CONST robtarget Target_880_2:=[[140.236685187,109.466342423,0],[0,-0.707106781,0.707106781,0],[-1,-1,0,1],[9E+09,9E+09,9E+09,9E+09,9E+09,9E+09]];
    CONST robtarget Target_890_2:=[[117.418637849,109.454015007,0],[0,-0.707106781,0.707106781,0],[-1,-1,0,1],[9E+09,9E+09,9E+09,9E+09,9E+09,9E+09]];
    CONST robtarget Target_940_2:=[[150.283504114,128.956035202,17.783725507],[0,-0.707106781,0.707106781,0],[-1,-1,0,1],[9E+09,9E+09,9E+09,9E+09,9E+09,9E+09]];
    CONST robtarget Target_910_2:=[[150.283529368,128.955987394,0],[0,-0.707106781,0.707106781,0],[-1,-1,0,1],[9E+09,9E+09,9E+09,9E+09,9E+09,9E+09]];
    CONST robtarget Target_920_2:=[[150.283529368,108.443166881,0],[0,-0.707106781,0.707106781,0],[-1,-1,0,1],[9E+09,9E+09,9E+09,9E+09,9E+09,9E+09]];
    CONST robtarget Target_930_2:=[[170.106014575,108.443166881,0],[0,-0.707106781,0.707106781,0],[-1,-1,0,1],[9E+09,9E+09,9E+09,9E+09,9E+09,9E+09]];
    CONST robtarget Target_950_2:=[[170.105997965,108.443230949,17.745858799],[0.000000043,-0.707106776,0.707106786,0.000000052],[-1,-1,0,1],[9E+09,9E+09,9E+09,9E+09,9E+09,9E+09]];
    CONST robtarget Target_980:=[[745.19998539,63.555998518,648.614999447],[0.403058195,0.127083777,0.864361092,0.272532031],[-1,0,0,0],[9E+09,9E+09,9E+09,9E+09,9E+09,9E+09]];
    TASK PERS wobjdata WorkPastel:=[FALSE,TRUE,"",[[700,297.348037667,137.083427328],[0.707046202,0.009255742,0.009255742,-0.707046202]],[[0,0,0],[1,0,0,0]]];
    TASK PERS wobjdata WorkPastel_2:=[FALSE,TRUE,"",[[663.397,-100,66.603],[0.683919377,0.179594782,-0.179594782,-0.683919377]],[[0,0,0],[1,0,0,0]]];
    CONST robtarget HomeRobot:=[[745.19998539,63.555998518,648.614999447],[0.403058195,0.127083777,0.864361092,0.272532031],[-1,0,0,0],[9E+09,9E+09,9E+09,9E+09,9E+09,9E+09]];
    CONST robtarget mantHerr:=[[494.621080465,494.792087576,971.864826811],[0.624444846,-0.306019376,0.699247952,0.165750044],[0,0,-1,0],[9E+09,9E+09,9E+09,9E+09,9E+09,9E+09]];
    CONST robtarget Target_970:=[[613.91794523,63.555999404,458.442114072],[0.041600547,0.221703595,0.952809214,0.203153911],[-1,0,0,0],[9E+09,9E+09,9E+09,9E+09,9E+09,9E+09]];
    CONST robtarget posMant:=[[458.575882142,-458.404912524,957.488606652],[0.61756941,0.262550436,0.653702432,-0.349783394],[-1,-1,-1,1],[9E+09,9E+09,9E+09,9E+09,9E+09,9E+09]];


!***********************************************************
    !
    ! M?dulo:  Module1
    !
    ! Descripción:
    !   <Introduzca la descripción aquí>
    !
    ! Autor: LENOVO
    !
    ! Versión: 1.0
    !
    !***********************************************************


    !***********************************************************
    !
    ! Procedimiento Main
    !
    !   Este es el punto de entrada de su programa
    !
    !***********************************************************
    PROC main()
        Inicio:
        IF DI_01=1 THEN
           Escribir;

        ENDIF
        IF DI_02=1 THEN
            Mantenimiento;
        ENDIF
        GOTO Inicio;
    ENDPROC

    LOCAL PROC Mantenimiento()
        Set DO_02;
        gomantHerr;
        Reset DO_02;
    ENDPROC

    LOCAL PROC Escribir()
        Set DO_01;
        goHome;
        goinicio;
        Fenix;
        Gio;
        Nic;
        goHome;
        Reset DO_01;
    ENDPROC

    LOCAL PROC Fenix()
        MoveL Home,v1000,z5,HerrG\WObj:=WorkPastel;
        MoveL Target_110,v500,z5,HerrG\WObj:=WorkPastel;
        MoveL Target_140,v100,z5,HerrG\WObj:=WorkPastel;
        MoveL Target_150,v100,z5,HerrG\WObj:=WorkPastel;
        MoveL Target_160,v100,z5,HerrG\WObj:=WorkPastel;
        MoveL Target_170,v100,z5,HerrG\WObj:=WorkPastel;
        MoveL Target_180,v100,z5,HerrG\WObj:=WorkPastel;
        MoveL Target_190,v100,z5,HerrG\WObj:=WorkPastel;
        MoveL Target_200,v100,z5,HerrG\WObj:=WorkPastel;
        MoveL Target_210,v100,z5,HerrG\WObj:=WorkPastel;
        MoveL Target_220,v100,z5,HerrG\WObj:=WorkPastel;
        MoveL Target_230,v100,z5,HerrG\WObj:=WorkPastel;
        MoveL Target_240,v100,z5,HerrG\WObj:=WorkPastel;
        MoveL Target_250,v100,z5,HerrG\WObj:=WorkPastel;
        MoveL Target_260,v100,z5,HerrG\WObj:=WorkPastel;
        MoveL Target_270,v100,z5,HerrG\WObj:=WorkPastel;
        MoveL Target_280,v100,z5,HerrG\WObj:=WorkPastel;
        MoveL Target_290,v100,z5,HerrG\WObj:=WorkPastel;
        MoveL Target_300,v100,z5,HerrG\WObj:=WorkPastel;
        MoveL Home,v500,z5,HerrG\WObj:=WorkPastel;
    ENDPROC
    LOCAL PROC G()
        MoveL Home,v1000,z5,HerrG\WObj:=WorkPastel;
        MoveL Target_960,v1000,z5,HerrG\WObj:=WorkPastel;
        MoveL Target_310,v100,z5,HerrG\WObj:=WorkPastel;
        MoveL Target_320,v100,z5,HerrG\WObj:=WorkPastel;
        MoveL Target_330,v100,z5,HerrG\WObj:=WorkPastel;
        MoveL Target_340,v100,z5,HerrG\WObj:=WorkPastel;
        MoveL Target_350,v100,z5,HerrG\WObj:=WorkPastel;
        MoveL Target_360,v100,z5,HerrG\WObj:=WorkPastel;
        MoveL Target_370,v100,z5,HerrG\WObj:=WorkPastel;
        MoveL Target_380,v100,z5,HerrG\WObj:=WorkPastel;
    ENDPROC
    LOCAL PROC I()
        MoveL Target_390,v100,z5,HerrG\WObj:=WorkPastel;
        MoveL Target_410,v100,z5,HerrG\WObj:=WorkPastel;
        MoveL Target_400,v100,z5,HerrG\WObj:=WorkPastel;
        MoveL Target_420,v100,z5,HerrG\WObj:=WorkPastel;
    ENDPROC
    LOCAL PROC O()
        MoveL Target_480,v100,z5,HerrG\WObj:=WorkPastel;
        MoveL Target_470,v100,z5,HerrG\WObj:=WorkPastel;
        MoveL Target_440,v100,z5,HerrG\WObj:=WorkPastel;
        MoveL Target_450,v100,z5,HerrG\WObj:=WorkPastel;
        MoveL Target_460,v100,z5,HerrG\WObj:=WorkPastel;
        MoveL Target_470,v100,z5,HerrG\WObj:=WorkPastel;
        MoveL Target_480,v100,z5,HerrG\WObj:=WorkPastel;
    ENDPROC
    LOCAL PROC V()
        MoveL Target_530,v100,z5,HerrG\WObj:=WorkPastel;
        MoveL Target_490,v100,z5,HerrG\WObj:=WorkPastel;
        MoveL Target_500,v100,z5,HerrG\WObj:=WorkPastel;
        MoveL Target_520,v100,z5,HerrG\WObj:=WorkPastel;
        MoveL Target_510,v100,z5,HerrG\WObj:=WorkPastel;
        MoveL Target_540,v100,z5,HerrG\WObj:=WorkPastel;
    ENDPROC
    LOCAL PROC A()
        MoveL Target_590,v1000,z5,HerrG\WObj:=WorkPastel;
        MoveL Target_550,v500,z5,HerrG\WObj:=WorkPastel;
        MoveL Target_560,v100,z5,HerrG\WObj:=WorkPastel;
        MoveL Target_570,v100,z5,HerrG\WObj:=WorkPastel;
        MoveL Target_580,v100,z5,HerrG\WObj:=WorkPastel;
        MoveL Target_600,v500,z5,HerrG\WObj:=WorkPastel;
    ENDPROC
    PROC Gio()
        G;
        I;
        O;
        V;
        A;
    ENDPROC
    PROC Inclinada()
        MoveJ Home_2,v1000,z5,HerrG\WObj:=WorkPastel_2;
        MoveL Target_110_2,v100,z5,HerrG\WObj:=WorkPastel_2;
        MoveL Target_140_2,v100,z5,HerrG\WObj:=WorkPastel_2;
        MoveL Target_150_2,v100,z5,HerrG\WObj:=WorkPastel_2;
        MoveL Target_160_2,v100,z5,HerrG\WObj:=WorkPastel_2;
        MoveL Target_170_2,v100,z5,HerrG\WObj:=WorkPastel_2;
        MoveL Target_180_2,v100,z5,HerrG\WObj:=WorkPastel_2;
        MoveL Target_190_2,v100,z5,HerrG\WObj:=WorkPastel_2;
        MoveL Target_200_2,v100,z5,HerrG\WObj:=WorkPastel_2;
        MoveL Target_210_2,v100,z5,HerrG\WObj:=WorkPastel_2;
        MoveL Target_220_2,v100,z5,HerrG\WObj:=WorkPastel_2;
        MoveL Target_230_2,v100,z5,HerrG\WObj:=WorkPastel_2;
        MoveL Target_240_2,v100,z5,HerrG\WObj:=WorkPastel_2;
        MoveL Target_250_2,v100,z5,HerrG\WObj:=WorkPastel_2;
        MoveL Target_260_2,v100,z5,HerrG\WObj:=WorkPastel_2;
        MoveL Target_270_2,v100,z5,HerrG\WObj:=WorkPastel_2;
        MoveL Target_280_2,v100,z5,HerrG\WObj:=WorkPastel_2;
        MoveL Target_290_2,v100,z5,HerrG\WObj:=WorkPastel_2;
        MoveL Target_300_2,v100,z5,HerrG\WObj:=WorkPastel_2;
        MoveL Home_2,v1000,z5,HerrG\WObj:=WorkPastel_2;
        MoveL Target_310_2,v100,z1,HerrG\WObj:=WorkPastel_2;
        MoveL Target_320_2,v100,z5,HerrG\WObj:=WorkPastel_2;
        MoveL Target_330_2,v100,z5,HerrG\WObj:=WorkPastel_2;
        MoveL Target_340_2,v100,z5,HerrG\WObj:=WorkPastel_2;
        MoveL Target_350_2,v100,z5,HerrG\WObj:=WorkPastel_2;
        MoveL Target_360_2,v100,z5,HerrG\WObj:=WorkPastel_2;
        MoveL Target_370_2,v100,z5,HerrG\WObj:=WorkPastel_2;
        MoveL Target_380_2,v100,z5,HerrG\WObj:=WorkPastel_2;
        MoveL Target_390_2,v100,z5,HerrG\WObj:=WorkPastel_2;
        MoveL Target_410_2,v100,z5,HerrG\WObj:=WorkPastel_2;
        MoveL Target_400_2,v100,z5,HerrG\WObj:=WorkPastel_2;
        MoveL Target_420_2,v100,z5,HerrG\WObj:=WorkPastel_2;
        MoveL Target_480_2,v100,z5,HerrG\WObj:=WorkPastel_2;
        MoveL Target_470_2,v100,z5,HerrG\WObj:=WorkPastel_2;
        MoveL Target_440_2,v100,z5,HerrG\WObj:=WorkPastel_2;
        MoveL Target_450_2,v100,z5,HerrG\WObj:=WorkPastel_2;
        MoveL Target_460_2,v100,z5,HerrG\WObj:=WorkPastel_2;
        MoveL Target_470_2,v100,z5,HerrG\WObj:=WorkPastel_2;
        MoveL Target_480_2,v100,z5,HerrG\WObj:=WorkPastel_2;
        MoveL Target_530_2,v100,z5,HerrG\WObj:=WorkPastel_2;
        MoveL Target_490_2,v100,z5,HerrG\WObj:=WorkPastel_2;
        MoveL Target_500_2,v100,z5,HerrG\WObj:=WorkPastel_2;
        MoveL Target_520_2,v100,z5,HerrG\WObj:=WorkPastel_2;
        MoveL Target_510_2,v100,z5,HerrG\WObj:=WorkPastel_2;
        MoveL Target_540_2,v100,z5,HerrG\WObj:=WorkPastel_2;
        MoveL Target_590_2,v100,z5,HerrG\WObj:=WorkPastel_2;
        MoveL Target_550_2,v100,z5,HerrG\WObj:=WorkPastel_2;
        MoveL Target_560_2,v100,z5,HerrG\WObj:=WorkPastel_2;
        MoveL Target_570_2,v100,z5,HerrG\WObj:=WorkPastel_2;
        MoveL Target_580_2,v100,z5,HerrG\WObj:=WorkPastel_2;
        MoveL Target_600_2,v100,z5,HerrG\WObj:=WorkPastel_2;
        MoveL Target_660_2,v100,z5,HerrG\WObj:=WorkPastel_2;
        MoveL Target_720_2,v100,z5,HerrG\WObj:=WorkPastel_2;
        MoveL Target_670_2,v100,z5,HerrG\WObj:=WorkPastel_2;
        MoveL Target_700_2,v100,z5,HerrG\WObj:=WorkPastel_2;
        MoveL Target_690_2,v100,z5,HerrG\WObj:=WorkPastel_2;
        MoveL Target_710_2,v100,z5,HerrG\WObj:=WorkPastel_2;
        MoveL Target_750_2,v100,z5,HerrG\WObj:=WorkPastel_2;
        MoveL Target_740_2,v100,z5,HerrG\WObj:=WorkPastel_2;
        MoveL Target_730_2,v100,z5,HerrG\WObj:=WorkPastel_2;
        MoveL Target_760_2,v100,z5,HerrG\WObj:=WorkPastel_2;
        MoveL Target_830_2,v100,z5,HerrG\WObj:=WorkPastel_2;
        MoveL Target_770_2,v100,z5,HerrG\WObj:=WorkPastel_2;
        MoveL Target_780_2,v100,z5,HerrG\WObj:=WorkPastel_2;
        MoveL Target_790_2,v100,z5,HerrG\WObj:=WorkPastel_2;
        MoveL Target_800_2,v100,z5,HerrG\WObj:=WorkPastel_2;
        MoveL Target_810_2,v100,z5,HerrG\WObj:=WorkPastel_2;
        MoveL Target_820_2,v100,z5,HerrG\WObj:=WorkPastel_2;
        MoveL Target_840_2,v100,z5,HerrG\WObj:=WorkPastel_2;
        MoveL Target_900_2,v100,z5,HerrG\WObj:=WorkPastel_2;
        MoveL Target_860_3,v100,z5,HerrG\WObj:=WorkPastel_2;
        MoveL Target_870_2,v100,z5,HerrG\WObj:=WorkPastel_2;
        MoveL Target_880_2,v100,z5,HerrG\WObj:=WorkPastel_2;
        MoveL Target_890_2,v100,z5,HerrG\WObj:=WorkPastel_2;
        MoveL Target_860_3,v100,z5,HerrG\WObj:=WorkPastel_2;
        MoveL Target_900_2,v100,z5,HerrG\WObj:=WorkPastel_2;
        MoveL Target_940_2,v100,z5,HerrG\WObj:=WorkPastel_2;
        MoveL Target_910_2,v100,z5,HerrG\WObj:=WorkPastel_2;
        MoveL Target_920_2,v100,z5,HerrG\WObj:=WorkPastel_2;
        MoveL Target_930_2,v100,z5,HerrG\WObj:=WorkPastel_2;
        MoveL Target_950_2,v100,z5,HerrG\WObj:=WorkPastel_2;
        MoveL Home_2,v100,z100,HerrG\WObj:=WorkPastel_2;
    ENDPROC
    PROC goHome()
        MoveJ Target_970,v600,z100,HerrG\WObj:=wobj0;
        MoveJ HomeRobot,v600,z100,HerrG\WObj:=wobj0;
    ENDPROC
    LOCAL PROC goinicio()
        MoveJ Target_650,v1000,z100,HerrG\WObj:=wobj0;
        MoveL Home,v1000,z100,HerrG\WObj:=WorkPastel;
    ENDPROC
    LOCAL PROC Nic()
        MoveL Target_660,v100,z5,HerrG\WObj:=WorkPastel;
        MoveL Target_720,v100,z5,HerrG\WObj:=WorkPastel;
        MoveL Target_670,v100,z5,HerrG\WObj:=WorkPastel;
        MoveL Target_680,v100,z5,HerrG\WObj:=WorkPastel;
        MoveL Target_700,v100,z5,HerrG\WObj:=WorkPastel;
        MoveL Target_690,v100,z5,HerrG\WObj:=WorkPastel;
        MoveL Target_710,v100,z5,HerrG\WObj:=WorkPastel;
        MoveL Target_750,v100,z5,HerrG\WObj:=WorkPastel;
        MoveL Target_740,v100,z5,HerrG\WObj:=WorkPastel;
        MoveL Target_730,v100,z5,HerrG\WObj:=WorkPastel;
        MoveL Target_760,v100,z5,HerrG\WObj:=WorkPastel;
        MoveL Target_830,v100,z5,HerrG\WObj:=WorkPastel;
        MoveL Target_770,v100,z5,HerrG\WObj:=WorkPastel;
        MoveL Target_780,v100,z5,HerrG\WObj:=WorkPastel;
        MoveL Target_790,v100,z5,HerrG\WObj:=WorkPastel;
        MoveL Target_800,v100,z5,HerrG\WObj:=WorkPastel;
        MoveL Target_810,v100,z5,HerrG\WObj:=WorkPastel;
        MoveL Target_820,v100,z5,HerrG\WObj:=WorkPastel;
        MoveL Target_840,v100,z5,HerrG\WObj:=WorkPastel;
        MoveL Target_900,v100,z5,HerrG\WObj:=WorkPastel;
        MoveL Target_860,v100,z5,HerrG\WObj:=WorkPastel;
        MoveL Target_870,v100,z5,HerrG\WObj:=WorkPastel;
        MoveL Target_880,v100,z5,HerrG\WObj:=WorkPastel;
        MoveL Target_890,v100,z5,HerrG\WObj:=WorkPastel;
        MoveL Target_860,v100,z5,HerrG\WObj:=WorkPastel;
        MoveL Target_900,v100,z5,HerrG\WObj:=WorkPastel;
        MoveL Target_940,v100,z5,HerrG\WObj:=WorkPastel;
        MoveL Target_910,v100,z5,HerrG\WObj:=WorkPastel;
        MoveL Target_920,v100,z5,HerrG\WObj:=WorkPastel;
        MoveL Target_930,v100,z5,HerrG\WObj:=WorkPastel;
        MoveL Target_950,v100,z5,HerrG\WObj:=WorkPastel;
    ENDPROC
    LOCAL PROC gomantHerr()
        MoveJ Target_970,v200,z50,HerrG\WObj:=wobj0;
        MoveJ posMant,v500,z50,HerrG\WObj:=wobj0;
    ENDPROC
ENDMODULE
